// TIA Portal V19 export
FUNCTION "FC_LadTest" : Void   // FC100, LAD
{ S7_Optimized_Access := 'TRUE' }
VERSION : 0.1
// stored: AutoNumber false, IsIECCheckEnabled false, SetENOAutomatically false
BEGIN

REGION Network 1
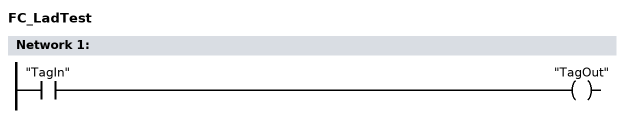
   RUNG wire#powerrail
      Contact( "TagIn" )
      Coil( "TagOut" )
   END_RUNG
   // the same network as SCL:
   "TagOut" := "TagIn";
END_REGION
END_FUNCTION
